// TIA Portal V15.1 export
// export: Created 2024-06-21T08:41:11.9176516Z, ExportSetting WithDefaults, DisplayName Totally Integrated Automation Portal, DisplayVersion V15.1 Update 5, DisplayName TIA Portal Openness, DisplayVersion V15.1 Update 5, DisplayName SINAMICS Startdrive Advanced, DisplayVersion V15.1, DisplayName G130, G150, S120, S150, SINAMICS MV, S210, DisplayVersion V15.1, DisplayName G110M, G120, G120C, G120D, G120P, DisplayVersion V15.1, DisplayName STEP 7 Professional, DisplayVersion V15.1 Update 5, DisplayName STEP 7 Safety, DisplayVersion V15.1, DisplayName WinCC Professional, DisplayVersion V15.1 Update 5, DisplayName SIMATIC Visualization Architect, DisplayVersion V15.1
FUNCTION_BLOCK "LGBCheckPipes"   // FB6669, SCL
TITLE = LBodyTypeSimSub
{ S7_Optimized_Access := 'TRUE' }
AUTHOR : IMTECH
VERSION : 1.0
// stored: AutoNumber false, IsIECCheckEnabled false, IsRetainMemResEnabled false, MemoryReserve 100, SetENOAutomatically False, UDAEnableTagReadback false
   VAR_INPUT
      I_CheckPipes { ExternalAccessible := 'False'; ExternalVisible := 'False'; ExternalWritable := 'False'} : Bool;   // Check if pipes are OK
      I_TopCoatColour { ExternalAccessible := 'False'; ExternalVisible := 'False'; ExternalWritable := 'False'} : Int;   // Top Coat Colour
      I_Spare1ColorCode { ExternalAccessible := 'False'; ExternalVisible := 'False'; ExternalWritable := 'False'} : Int;   // Spare colour Code
      I_Spare2ColorCode { ExternalAccessible := 'False'; ExternalVisible := 'False'; ExternalWritable := 'False'} : Int;   // Spare colour Code
      I_Spare3ColorCode { ExternalAccessible := 'False'; ExternalVisible := 'False'; ExternalWritable := 'False'} : Int;   // Spare colour Code
      I_Spare4ColorCode { ExternalAccessible := 'False'; ExternalVisible := 'False'; ExternalWritable := 'False'} : Int;   // Spare colour Code
      I_Spare5ColorCode { ExternalAccessible := 'False'; ExternalVisible := 'False'; ExternalWritable := 'False'} : Int;   // Spare colour Code
   END_VAR
   VAR_OUTPUT
      O_Ibc1OK { ExternalAccessible := 'False'; ExternalVisible := 'False'; ExternalWritable := 'False'} : Bool;   // IBC top coat 1
      O_Obc11Ok { ExternalAccessible := 'False'; ExternalVisible := 'False'; ExternalWritable := 'False'} : Bool;   // OBC1 top coat 1
      O_Obc12Ok { ExternalAccessible := 'False'; ExternalVisible := 'False'; ExternalWritable := 'False'} : Bool;   // OBC2 top coat 1
      O_TC1Ok { ExternalAccessible := 'False'; ExternalVisible := 'False'; ExternalWritable := 'False'} : Bool;   // Top coat 1 Ok
      O_TC1Nok { ExternalAccessible := 'False'; ExternalVisible := 'False'; ExternalWritable := 'False'} : Bool;   // Top coat 1 Nok
      O_Ibc2OK { ExternalAccessible := 'False'; ExternalVisible := 'False'; ExternalWritable := 'False'} : Bool;   // IBC top coat 2
      O_Obc21Ok { ExternalAccessible := 'False'; ExternalVisible := 'False'; ExternalWritable := 'False'} : Bool;   // OBC1 top coat 2
      O_Obc22Ok { ExternalAccessible := 'False'; ExternalVisible := 'False'; ExternalWritable := 'False'} : Bool;   // OBC2 top coat 2
      O_TC2Ok { ExternalAccessible := 'False'; ExternalVisible := 'False'; ExternalWritable := 'False'} : Bool;   // Top coat 2 Ok
      O_TC2Nok { ExternalAccessible := 'False'; ExternalVisible := 'False'; ExternalWritable := 'False'} : Bool;   // Top coat 2 Nok
   END_VAR
   VAR_IN_OUT
      IO_Pipe : Array[1..50] of "TCPipe";   // Pipe data
      IO_ValveData : Array[1..50] of "TCValve";   // Pipe valve data
      IO_RecipeData : Array[1..35] of "TCRecipe";   // Recipe data
      IO_RecipeDataCalculate : Array[1..35] of "TCRecipe";   // Recipe data calculate
   END_VAR
   VAR
      Ibc1OK { ExternalAccessible := 'False'; ExternalVisible := 'False'; ExternalWritable := 'False'} : Bool;   // IBC top coat 1
      Obc11Ok { ExternalAccessible := 'False'; ExternalVisible := 'False'; ExternalWritable := 'False'} : Bool;   // OBC1 top coat 1
      Obc12Ok { ExternalAccessible := 'False'; ExternalVisible := 'False'; ExternalWritable := 'False'} : Bool;   // OBC2 top coat 1
      Ibc2OK { ExternalAccessible := 'False'; ExternalVisible := 'False'; ExternalWritable := 'False'} : Bool;   // IBC top coat 2
      Obc21Ok { ExternalAccessible := 'False'; ExternalVisible := 'False'; ExternalWritable := 'False'} : Bool;   // OBC1 top coat 2
      Obc22Ok { ExternalAccessible := 'False'; ExternalVisible := 'False'; ExternalWritable := 'False'} : Bool;   // OBC2 top coat 2
      Index { ExternalAccessible := 'False'; ExternalVisible := 'False'; ExternalWritable := 'False'} : Int;
      IndexRecipe { ExternalAccessible := 'False'; ExternalVisible := 'False'; ExternalWritable := 'False'} : Int;
      IndexIbcColorCode { ExternalAccessible := 'False'; ExternalVisible := 'False'; ExternalWritable := 'False'} : Int;
      IndexObc1ColorCode { ExternalAccessible := 'False'; ExternalVisible := 'False'; ExternalWritable := 'False'} : Int;
      IndexObc2ColorCode { ExternalAccessible := 'False'; ExternalVisible := 'False'; ExternalWritable := 'False'} : Int;
      IbcColorCode { ExternalAccessible := 'False'; ExternalVisible := 'False'; ExternalWritable := 'False'} : Int;
      Obc1ColorCode { ExternalAccessible := 'False'; ExternalVisible := 'False'; ExternalWritable := 'False'} : Int;
      Obc2ColorCode { ExternalAccessible := 'False'; ExternalVisible := 'False'; ExternalWritable := 'False'} : Int;
      ColorCodeNOK { ExternalAccessible := 'False'; ExternalVisible := 'False'; ExternalWritable := 'False'} : Bool;   // Colour Code NOK
   END_VAR
BEGIN
   //************************************
   //*                                  *
   //*             LOGIC FB             *
   //*                                  *
   //************************************

   // CLEAR bits
   #Ibc1OK := False;
   #Obc11Ok := False;
   #Obc12Ok := False;
   #Ibc2OK := False;
   #Obc21Ok := False;
   #Obc22Ok := False;
   #ColorCodeNOK := False;

   //Color code Not OK or Not existing
   IF #I_TopCoatColour = #I_Spare1ColorCode OR
       #I_TopCoatColour = #I_Spare2ColorCode OR
       #I_TopCoatColour = #I_Spare3ColorCode OR
       #I_TopCoatColour = #I_Spare4ColorCode OR
       #I_TopCoatColour = #I_Spare5ColorCode THEN
       #ColorCodeNOK := TRUE;
   END_IF;

   //Check pipe data
   IF #I_CheckPipes THEN
       //Find recipe
       FOR #IndexRecipe := 1 TO 35 DO
           IF #I_TopCoatColour = #IO_RecipeData[#IndexRecipe].TagColorCode THEN
               #IbcColorCode := #IO_RecipeData[#IndexRecipe].IBCColorCode;
               #Obc1ColorCode := #IO_RecipeData[#IndexRecipe].OBC1ColorCode;
               #Obc2ColorCode := #IO_RecipeData[#IndexRecipe].OBC2ColorCode;
               //Check IBC for TC1 and TC2
               FOR #IndexIbcColorCode := 1 TO 50 DO
                   IF #IbcColorCode = #IO_Pipe[#IndexIbcColorCode].ColorCode THEN
                       #Ibc1OK := #IO_ValveData[#IndexIbcColorCode].IBC1 = 2 OR #IO_ValveData[#IndexIbcColorCode].IBC1 = 4;
                       #Ibc2OK := #IO_ValveData[#IndexIbcColorCode].IBC2 = 2 OR #IO_ValveData[#IndexIbcColorCode].IBC2 = 4;
                       EXIT;
                   END_IF;
               END_FOR;
               //Check OBC1 for TC1 and TC2
               FOR #IndexObc1ColorCode := 1 TO 50 DO
                   IF #Obc1ColorCode = #IO_Pipe[#IndexObc1ColorCode].ColorCode THEN
                       #Obc11Ok := #IO_ValveData[#IndexObc1ColorCode].OBC11 = 2 OR #IO_ValveData[#IndexObc1ColorCode].OBC11 = 4;
                       #Obc21Ok := #IO_ValveData[#IndexObc1ColorCode].OBC21 = 2 OR #IO_ValveData[#IndexObc1ColorCode].OBC21 = 4;
                       EXIT;
                   END_IF;
               END_FOR;
               //Check OBC2 for TC1 and TC2
               IF #IO_RecipeDataCalculate[#IndexRecipe].ColorType = 1 THEN //Don't check OBC2 when colortype is 1
                   #Obc12Ok := True;
                   #Obc22Ok := True;
               ELSE
                   FOR #IndexObc2ColorCode := 1 TO 50 DO
                       IF #Obc2ColorCode = #IO_Pipe[#IndexObc2ColorCode].ColorCode THEN
                           #Obc12Ok := #IO_ValveData[#IndexObc2ColorCode].OBC12 = 2 OR #IO_ValveData[#IndexObc2ColorCode].OBC12 = 4;
                           #Obc22Ok := #IO_ValveData[#IndexObc2ColorCode].OBC22 = 2 OR #IO_ValveData[#IndexObc2ColorCode].OBC22 = 4;
                           EXIT;
                       END_IF;
                   END_FOR;
               END_IF;
               EXIT;
           END_IF;
       END_FOR;
   END_IF;

   // OUTPUT
   #O_Ibc1OK := #Ibc1OK OR #ColorCodeNOK;
   #O_Obc11Ok := #Obc11Ok OR #ColorCodeNOK;
   #O_Obc12Ok := #Obc12Ok OR #ColorCodeNOK;
   #O_TC1Ok := (#Ibc1OK AND #Obc11Ok AND #Obc12Ok) OR #ColorCodeNOK;
   #O_TC1Nok := NOT ((#Ibc1OK AND #Obc11Ok AND #Obc12Ok) OR #ColorCodeNOK) AND #I_CheckPipes;

   #O_Ibc2OK := #Ibc2OK  OR #ColorCodeNOK;
   #O_Obc21Ok := #Obc21Ok OR #ColorCodeNOK;
   #O_Obc22Ok := #Obc22Ok OR #ColorCodeNOK;
   #O_TC2Ok := (#Ibc2OK AND #Obc21Ok AND #Obc22Ok) OR #ColorCodeNOK;
   #O_TC2Nok := NOT ((#Ibc2OK AND #Obc21Ok AND #Obc22Ok) OR #ColorCodeNOK) AND #I_CheckPipes;
END_FUNCTION_BLOCK
